(* CODESYS project TANQUEE.project

Project tree, tasks and I/O mapping:
  Device : CODESYS Control Win V3, 3S - Smart Software Solutions GmbH, order no. 305021, version 3.5.11.30
    application Application
      libraries: Standard, * (System)
      task MainTask (cyclic, interval t#20ms, priority 1) calls PLC_PRG
      program PLC_PRG [LD]
*)

// Device/Application/PLC_PRG
PROGRAM PLC_PRG
VAR
	START : BOOL;       // INICIA O PROCESSO
    MV1 : BOOL;         // LIBERA O FLUXO DE AGUA NO TANQUE
	LT1 : BOOL;         // SENSOR DE NIVEL INICIAL DO TANQUE
    LT2 : BOOL;         // SENSOR DE NIVEL MEDIO DO TANQUE
    EST : BOOL;         // MOTOR DA ESTEIRA 
    LT3 : BOOL;         // SENSOR DO TOPO DO TANQUE
    STIR : BOOL;        // MOTOR PARA MISTURAR O CONTEUDO
    MV2 : BOOL;         // VALVULA DA SAIDA DE AGUA NOTANQUE
	P1: BOOL;
	P3: BOOL;
	P2: BOOL;
	P4: BOOL;
	TOF_1: TOF;
	ET1: TIME;
	AUX1 : BOOL;
	TON_1: TON;
	ET2: TIME;
	CTU_1: CTU;
	CV1: WORD;
	P5: BOOL;
	P6: BOOL;
	STOP: BOOL;
	AUX2: BOOL;
END_VAR
VAR // added by the converter: edge detectors and wires of the graphical bodies
    _rt1, _rt2, _rt3 : R_TRIG;
END_VAR

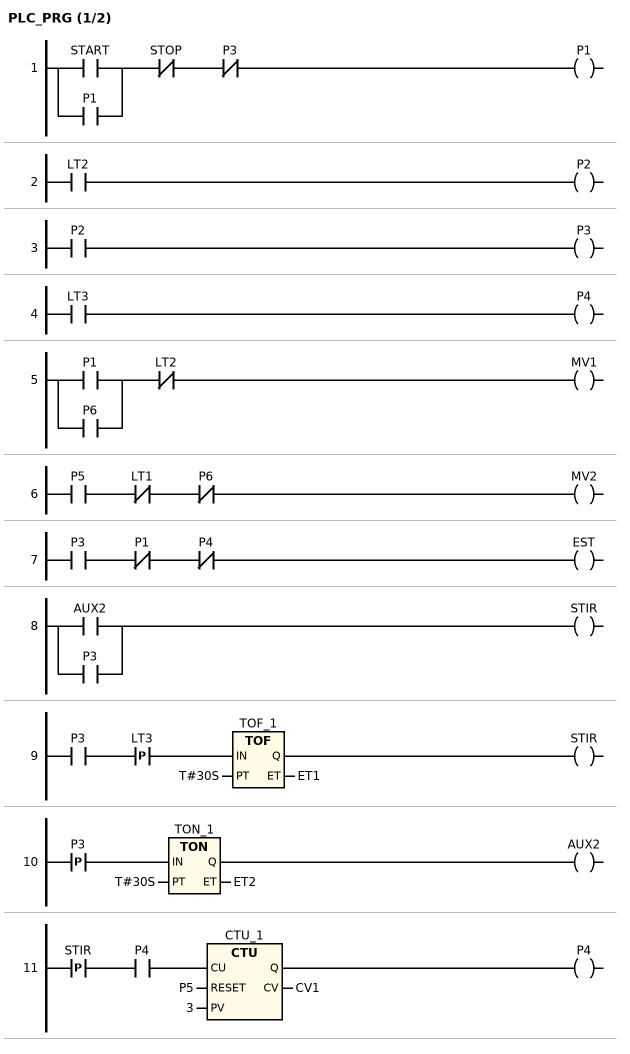
// NETWORK 1
P1 := (START OR P1) AND NOT STOP AND NOT P3;

// NETWORK 2
P2 := LT2;

// NETWORK 3
P3 := P2;

// NETWORK 4
P4 := LT3;

// NETWORK 5
MV1 := (P1 OR P6) AND NOT LT2;

// NETWORK 6
MV2 := P5 AND NOT LT1 AND NOT P6;

// NETWORK 7
EST := P3 AND NOT P1 AND NOT P4;

// NETWORK 8
STIR := AUX2 OR P3;

// NETWORK 9
_rt1(CLK := LT3);
TOF_1(IN := P3 AND _rt1.Q, PT := T#30S, ET => ET1); // TOF
STIR := TOF_1.Q;

// NETWORK 10
_rt2(CLK := P3);
TON_1(IN := _rt2.Q, PT := T#30S, ET => ET2); // TON
AUX2 := TON_1.Q;

// NETWORK 11
_rt3(CLK := STIR);
CTU_1(CU := _rt3.Q AND P4, RESET := P5, PV := 3, CV => CV1); // CTU
P4 := CTU_1.Q;

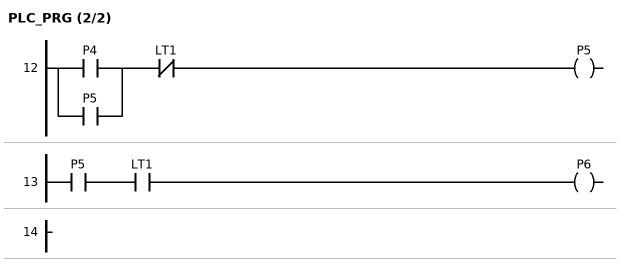
// NETWORK 12
P5 := (P4 OR P5) AND NOT LT1;

// NETWORK 13
P6 := P5 AND LT1;

// NETWORK 14

END_PROGRAM
